// TIA Portal V17 export
// export: Created 2025-04-11T04:54:22.9167246Z, ExportSetting WithDefaults, DisplayName Totally Integrated Automation Portal, DisplayVersion V17, DisplayName TIA Portal Openness, DisplayVersion V17, DisplayName TIA Portal Version Control Interface, DisplayVersion V17, DisplayName SINAMICS Startdrive Advanced, DisplayVersion V17, DisplayName SINAMICS Startdrive G130, G150, S120, S150, SINAMICS MV, S210, DisplayVersion V17, DisplayName SINAMICS Startdrive G110M, G120, G120C, G120D, G120P, G115D, DisplayVersion V17, DisplayName STEP 7 Professional, DisplayVersion V17, DisplayName STEP 7 Safety, DisplayVersion V17, DisplayName WinCC Advanced, DisplayVersion V17
TYPE "UDT_Modbus_Config"
// stored: IsFailsafeCompliant false
   STRUCT
      mbAddr : UInt;   // Modbus从站地址
      mode : USInt;   // 通信模式(0=读,1=写)
      dataAddr : UDInt;   // 数据地址
      dataLen : UInt;   // 数据长度
      instrument : DB_ANY;   // 数据块指针
   END_STRUCT;
END_TYPE
